SUBAPPLICATION Uebung_223_AX (* Standard IEC 61131-3 AUDI_FB_CTUD (Adapter Version, UDINT) *)
  (* Standard: 61131-3; Description: Copyright (c) 2026 Meisterschulen am Ostbahnhof This program and the accompanying materials are made available under the terms of the Eclipse Public License 2.0 which is available at https://www.eclipse.org/legal/epl-2.0/ SPDX-License-Identifier: EPL-2.0 *)
  (* Version 1.0, 2026-04-21, Franz Höpfinger, Meisterschulen am Ostbahnhof, initial API and implementation (Adapter version) *)
  PACKAGE Uebungen;
  IMPORT logiBUS::io::DI::logiBUS_DI::Input_I1;
  IMPORT logiBUS::io::DI::logiBUS_DI::Input_I2;
  IMPORT logiBUS::io::DI::logiBUS_DI::Input_I3;
  IMPORT logiBUS::io::DI::logiBUS_DI::Input_I4;
  IMPORT logiBUS::io::DQ::logiBUS_DO::Output_Q1;
  IMPORT logiBUS::io::DQ::logiBUS_DO::Output_Q2;
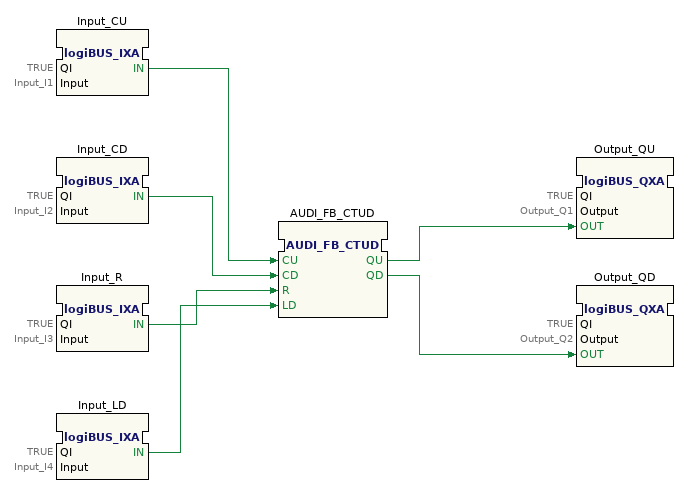
  FBS
    AUDI_FB_CTUD : adapter::iec61131_3::counters::AUDI_FB_CTUD;
    Input_CU : logiBUS::io::DI::logiBUS_IXA(QI := TRUE, Input := Input_I1);
    Input_CD : logiBUS::io::DI::logiBUS_IXA(QI := TRUE, Input := Input_I2);
    Input_R : logiBUS::io::DI::logiBUS_IXA(QI := TRUE, Input := Input_I3);
    Input_LD : logiBUS::io::DI::logiBUS_IXA(QI := TRUE, Input := Input_I4);
    Output_QU : logiBUS::io::DQ::logiBUS_QXA(QI := TRUE, Output := Output_Q1);
    Output_QD : logiBUS::io::DQ::logiBUS_QXA(QI := TRUE, Output := Output_Q2);
  END_FBS
  ADAPTER_CONNECTIONS
    Input_CU.IN TO AUDI_FB_CTUD.CU;
    Input_CD.IN TO AUDI_FB_CTUD.CD;
    Input_R.IN TO AUDI_FB_CTUD.R;
    Input_LD.IN TO AUDI_FB_CTUD.LD;
    AUDI_FB_CTUD.QU TO Output_QU.OUT;
    AUDI_FB_CTUD.QD TO Output_QD.OUT;
  END_CONNECTIONS
END_SUBAPPLICATION
